// TIA Portal V21 export
VAR_GLOBAL   // PLC tag table "K_TipoPortata"
END_VAR
VAR_GLOBAL CONSTANT   // user constants
   K_TipoPortataDaImpulso : Int := 0;
   K_TipoPortataDaAnalogica : Int := 1;
END_VAR
